// TIA Portal V17 export
// export: Created 2025-11-19T10:30:00.000Z, ExportSetting WithDefaults, DisplayName Totally Integrated Automation Portal, DisplayVersion V17
FUNCTION_BLOCK "FB_PID_Controller"   // FB20, SCL
{ S7_Optimized_Access := 'TRUE' }
AUTHOR : Control Systems
FAMILY : Controllers
NAME : PID Controller
VERSION : 2.1
// stored: AutoNumber true, IsIECCheckEnabled true
   VAR_INPUT
      Setpoint : Real;
      ProcessValue : Real;
      Kp : Real;
      Ki : Real;
      Kd : Real;
      Enable : Bool;
   END_VAR
   VAR_OUTPUT
      ControlOutput : Real;
      Error : Real;
   END_VAR
   VAR
      IntegralSum : Real;
      LastError : Real;
      Initialized : Bool;
   END_VAR
   VAR_TEMP
      PropTerm : Real;
      IntTerm : Real;
      DiffTerm : Real;
   END_VAR
BEGIN
// PID Control Algorithm - BUGGY
// BUGS: Inverted error sign, no input validation, no pre-windup anti-windup, unbounded integral, inverted anti-windup limits, missing error reset, derivative kick, no deadband, wrong anti-windup correction
   0.0 THEN0.0 THEN0.0 THEN0.0 THEN0.0 THEN0.0 THEN0.0 THEN0.00.00.0 THEN0.0;0.0;
          0.0;
          0.0;
           #IntegralSum :=0.0;
           #IntegralSum = 0.0;0.
END_FUNCTION_BLOCK
